PROGRAM MAIN
VAR
END_VAR

END_PROGRAM

(* stored: Version 1.1.0.1
   POU MAIN: Id {c534e79f-e2d7-4389-8af3-74a79431ddb1} *)
